FUNCTION_BLOCK sqlUpdateMaterial (* Tamplate for a simple Basic Function Block Type *)
  (* Standard: 61499-2 *)
  (* Version 0.0, 2018-01-05, 4DIAC-IDE, 4DIAC-Consortium *)
  (* Version 1.0, 2016-05-26, AZ, fortiss GmbH *)
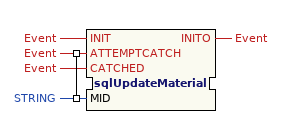
  EVENT_INPUT
    INIT; (* Initialization Request *)
    ATTEMPTCATCH WITH MID;
    CATCHED; (* Normal Execution Request *)
  END_EVENT
  EVENT_OUTPUT
    INITO; (* Initialization Confirm *)
  END_EVENT
  VAR_INPUT
    MID : STRING; (* Input event qualifier *)
  END_VAR
  VAR
    catchMid : STRING; (* Internal Variable *)
  END_VAR
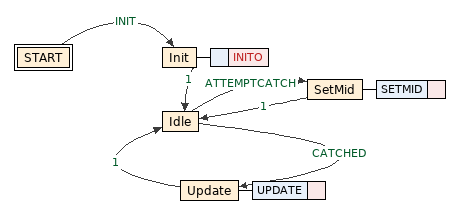
  EC_STATES
    START; (* Initial State *)
    Init : -> INITO; (* Initialization *)
    Idle;
    Update : UPDATE;
    SetMid : SETMID;
  END_STATES
  EC_TRANSITIONS
    START TO Init := INIT;
    Init TO Idle := 1;
    Idle TO Update := CATCHED;
    Update TO Idle := 1;
    Idle TO SetMid := ATTEMPTCATCH;
    SetMid TO Idle := 1;
  END_TRANSITIONS
  ALGORITHM UPDATE IN ST: (* new algorithm *)

  END_ALGORITHM
  ALGORITHM SETMID IN ST: (* new algorithm *)
catchMid := MID;
  END_ALGORITHM
END_FUNCTION_BLOCK
